FUNCTION WRITE_ANY_DATE : BOOL
VAR_INPUT
    ptr: POINTER TO DATE;
    val: DATE;
END_VAR

ptr^ := val;

END_FUNCTION

(* stored: Version 1.1.0.1, ProductVersion 3.1.4022.9
   POU WRITE_ANY_DATE: Id {79d90978-55d9-4c8a-9385-a65057de0645}, SpecialFunc None *)
